// Mitsubishi GX Works2 project: EX2_GROUP21   PLC: FX3G

// global labels: Global1
VAR_GLOBAL
  Emergency AT X005 : BOOL;
  Enough_Materials AT M1 : BOOL;
  Storage_Packs AT D1100 : REAL;
END_VAR
VAR_GLOBAL CONSTANT
  Esroni : REAL := 10.0;
END_VAR
VAR_GLOBAL
  Packs_Display AT D8282 : INT;
  Start_Day AT X007 : BOOL;
  AI_GumType AT D8280 : INT;
  Init_raspberry AT D1150 : REAL;
  Stock_Raspberry AT D2500 : REAL;
  Stock_Lemon AT D2200 : REAL;
  Init_Stabilizer AT D1130 : REAL;
  Stock_Stabilizer AT D2300 : REAL;
  Init_Gummies AT D1140 : REAL;
  Stock_Gummies AT D2400 : REAL;
  Start_Production AT X001 : BOOL;
  Enough_Raspberry AT M9 : BOOL;
  Enough_Lemon AT M10 : BOOL;
  Enough_Stabilizer AT M11 : BOOL;
  Enough_Gummies AT M12 : BOOL;
  Day_Lamp AT Y007 : BOOL;
  GumType_Sempeld AT D3000 : REAL;
  Type_Regular AT M3 : BOOL;
  Type_Premium AT M2 : BOOL;
  Step_Preparation AT M4 : BOOL;
  Prep_Timer AT TC0 : BOOL;
  Stop_Blend AT M14 : BOOL;
  Prep_Counter AT TS0 : BOOL;
  Prep_Lamp AT Y000 : BOOL;
  Start_Cooling AT X002 : BOOL;
  Stop_Prep AT M13 : BOOL;
  Step_Cooling AT M5 : BOOL;
  Stop_Cooling AT TS1 : BOOL;
  Temp_OK AT X003 : BOOL;
  Cooling_Timer AT TC1 : BOOL;
  Cool_Time AT K80 : INT;
  Cooling_Lamp AT Y002 : BOOL;
  Step_Mixing AT M6 : BOOL;
  Blink_Bit AT M8 : BOOL;
  Blink_Time AT K10 : INT;
  Mix_LampA AT Y005 : BOOL;
  Blink_TimerB AT TC3 : BOOL;
  Blink_TimerA AT TC2 : BOOL;
  Stop_BlinkingB AT TS3 : BOOL;
  Stop_BlinkingA AT TS2 : BOOL;
  Mix_LampB AT Y006 : BOOL;
  Mix_Timer_R AT TC4 : BOOL;
  Regular_Mixing_Time AT K30 : INT;
  Mix_Timer_P AT TC5 : BOOL;
  Premium_Mixing_Time AT K50 : INT;
  Mixing_Timer_R AT TS4 : BOOL;
  Mixing_Timer_P AT TS5 : BOOL;
END_VAR
VAR_GLOBAL CONSTANT
  Constant280 : REAL := 280.0;
  Constant400 : REAL := 400.0;
END_VAR
VAR_GLOBAL
  Start_Packing AT M15 : BOOL;
END_VAR
VAR_GLOBAL CONSTANT
  Add_Pack : REAL := 1.0;
  LE_K5 : REAL := 5.0;
  GT_K6 : REAL := 6.0;
  GT_K10 : REAL := 10.0;
  ReqRaspberry : REAL := 385.0;
  ReqLemon : REAL := 665.0;
  ReqStabilizer : REAL := 210.0;
  ReqGummies : REAL := 70.0;
END_VAR
VAR_GLOBAL
  GumType_Final AT D3010 : REAL;
END_VAR
VAR_GLOBAL CONSTANT
  LE_K10 : REAL := 10.0;
END_VAR
VAR_GLOBAL
  Type_R AT M16 : BOOL;
END_VAR
VAR_GLOBAL CONSTANT
  ZeroStartDay : REAL;
END_VAR
VAR_GLOBAL
  Init_Lemon AT D1120 : REAL;
END_VAR
VAR_GLOBAL CONSTANT
  Respberry_280 : REAL := 280.0;
  Gummies_28 : REAL := 28.0;
  Stebilizer_105 : REAL := 105.0;
  Lemon_455 : REAL := 455.0;
END_VAR
VAR_GLOBAL
  Sec_5 AT K50 : INT;
  Not_Active AT M17 : BOOL;
END_VAR

// task Task_01 (event TRUE, interval 0, priority 31): POU_01

PROGRAM POU_01
(* structured ladder/FBD written out as ST: instructions are called as NAME(EN, inputs, outputs); _pN, _eN, _tN stand for wires *)
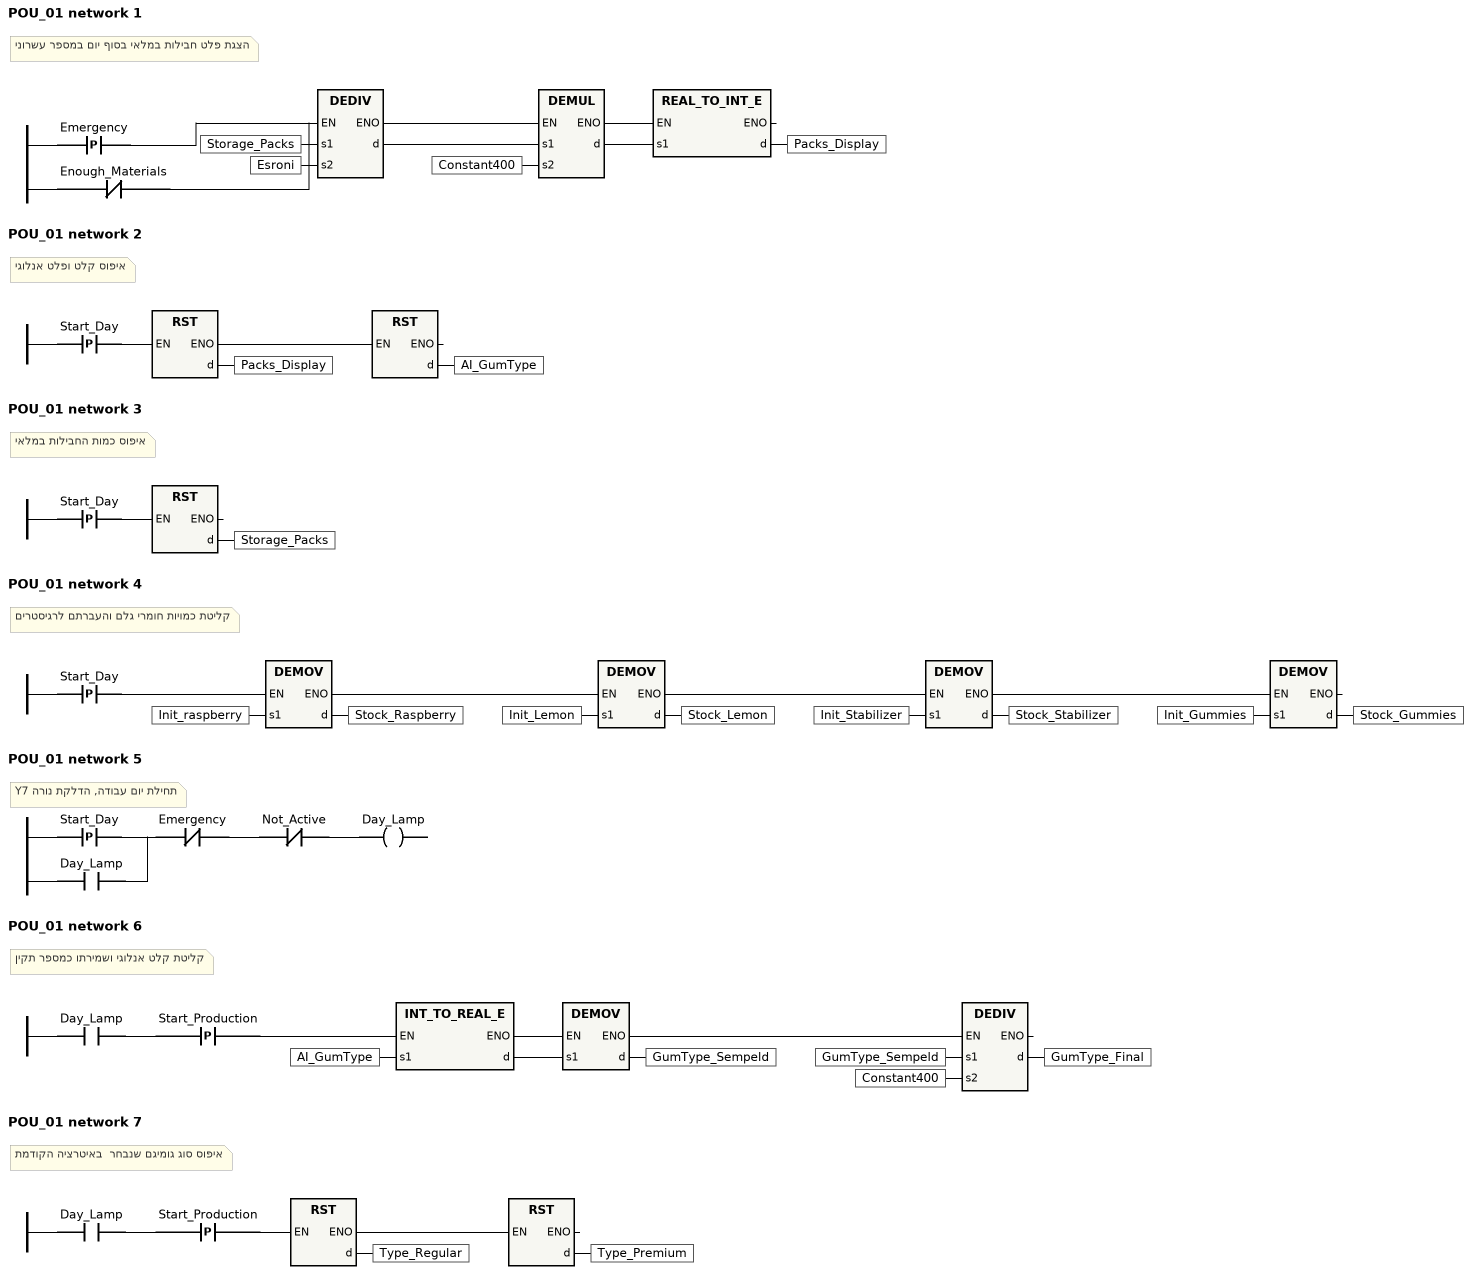
(* network 1 *)
(* הצגת פלט חבילות במלאי בסוף יום במספר עשרוני *)
_e2 := DEDIV(LDP(TRUE, Emergency) OR (NOT Enough_Materials), Storage_Packs, Esroni, _t1);
_e4 := DEMUL(_e2, _t1, Constant400, _t3);
REAL_TO_INT_E(_e4, _t3, Packs_Display);
(* network 2 *)
(* איפוס קלט ופלט אנלוגי *)
_e1 := RST(LDP(TRUE, Start_Day), Packs_Display);
RST(_e1, AI_GumType);
(* network 3 *)
(* איפוס כמות החבילות במלאי *)
RST(LDP(TRUE, Start_Day), Storage_Packs);
(* network 4 *)
(* קליטת כמויות חומרי גלם והעברתם לרגיסטרים *)
_e1 := DEMOV(LDP(TRUE, Start_Day), Init_raspberry, Stock_Raspberry);
_e2 := DEMOV(_e1, Init_Lemon, Stock_Lemon);
_e3 := DEMOV(_e2, Init_Stabilizer, Stock_Stabilizer);
DEMOV(_e3, Init_Gummies, Stock_Gummies);
(* network 5 *)
(* תחילת יום עבודה, הדלקת נורה Y7 *)
Day_Lamp := ((LDP(TRUE, Start_Day) OR Day_Lamp) AND NOT Emergency) AND NOT Not_Active;
(* network 6 *)
(* קליטת קלט אנלוגי ושמירתו כמספר תקין *)
_e2 := INT_TO_REAL_E(Day_Lamp AND LDP(TRUE, Start_Production), AI_GumType, _t1);
_e3 := DEMOV(_e2, _t1, GumType_Sempeld);
DEDIV(_e3, GumType_Sempeld, Constant400, GumType_Final);
(* network 7 *)
(* איפוס סוג גומיגם שנבחר  באיטרציה הקודמת *)
_e1 := RST(Day_Lamp AND LDP(TRUE, Start_Production), Type_Regular);
RST(_e1, Type_Premium);
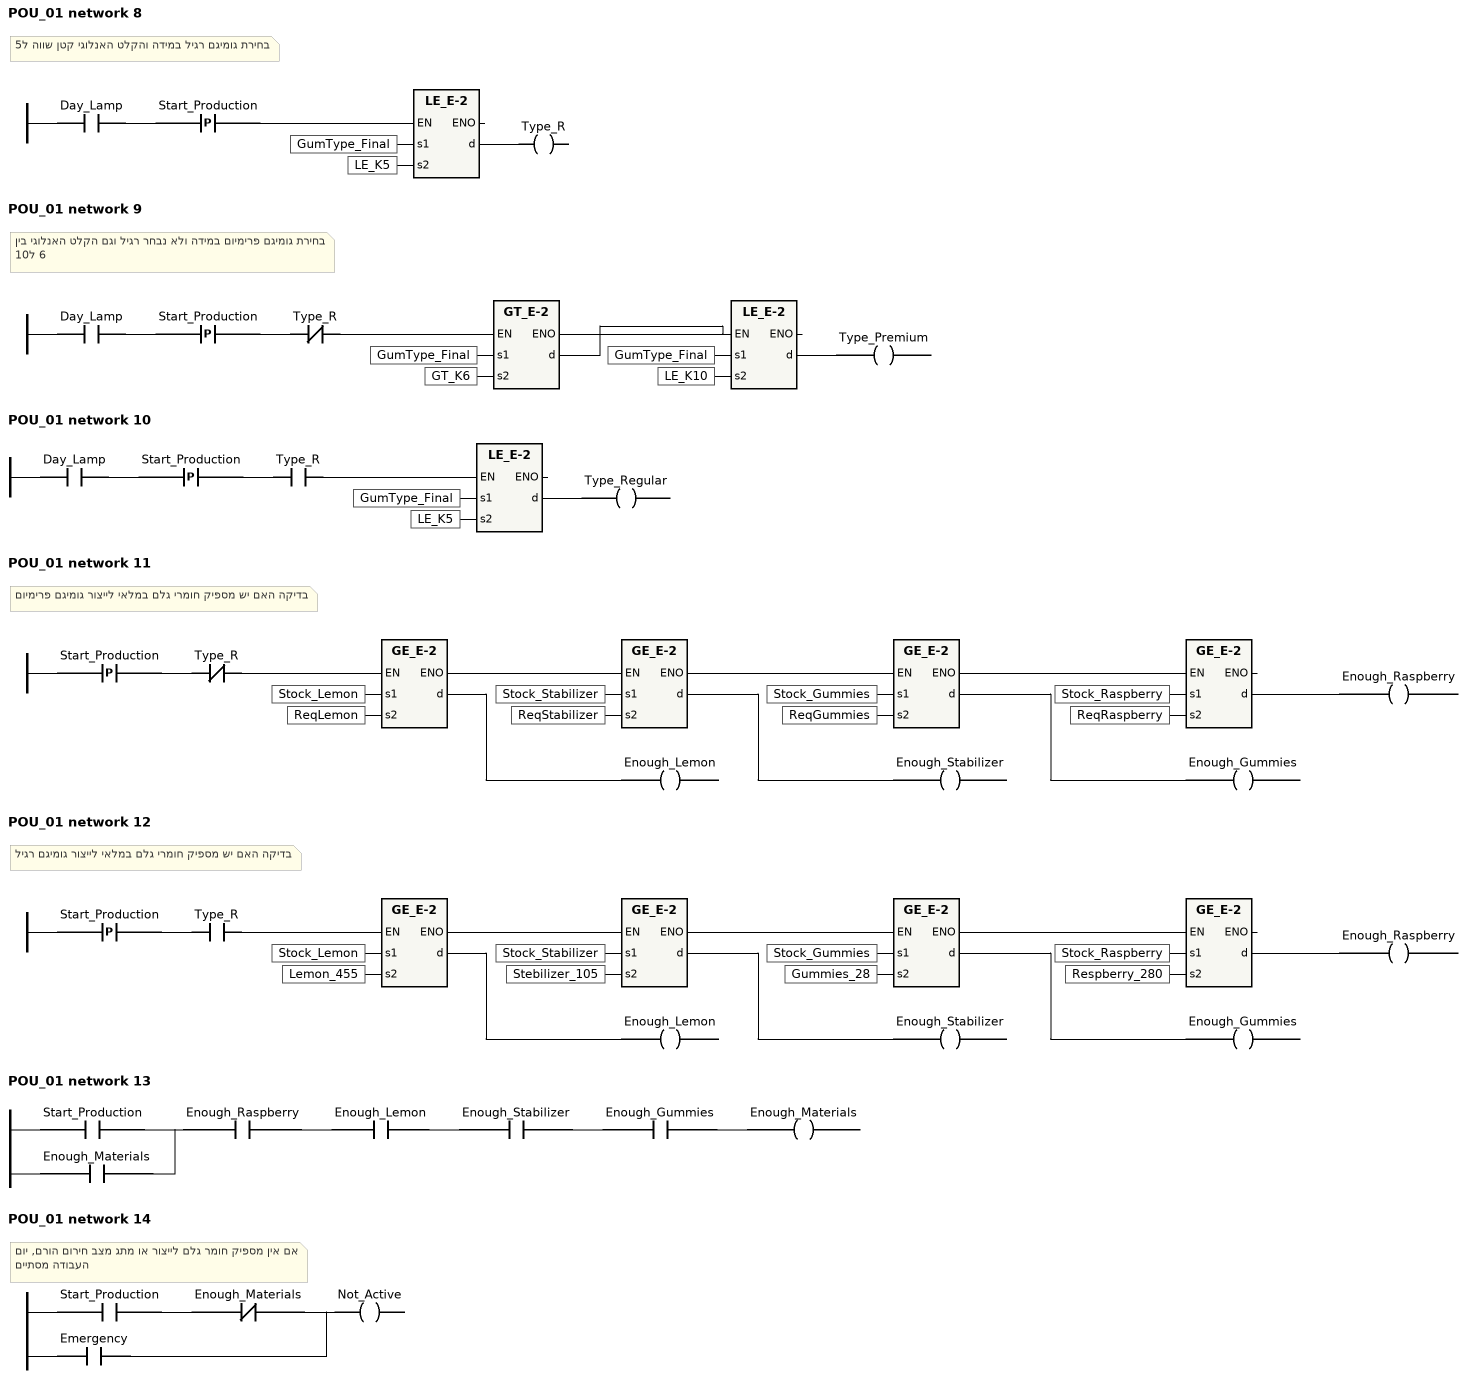
(* network 8 *)
(* בחירת גומיגם רגיל במידה והקלט האנלוגי קטן שווה ל5 *)
LE_E(Day_Lamp AND LDP(TRUE, Start_Production), GumType_Final, LE_K5, _t1);
Type_R := _t1;
(* network 9 *)
(* בחירת גומיגם פרימיום במידה ולא נבחר רגיל וגם הקלט האנלוגי בין 6 ל10 *)
_e2 := GT_E(Day_Lamp AND LDP(TRUE, Start_Production) AND NOT Type_R, GumType_Final, GT_K6, _t1);
LE_E(_e2 OR _t1, GumType_Final, LE_K10, _t3);
Type_Premium := _t3;
(* network 10 *)
LE_E(Day_Lamp AND LDP(TRUE, Start_Production) AND Type_R, GumType_Final, LE_K5, _t1);
Type_Regular := _t1;
(* network 11 *)
(* בדיקה האם יש מספיק חומרי גלם במלאי לייצור גומיגם פרימיום *)
_e2 := GE_E(LDP(TRUE, Start_Production) AND NOT Type_R, Stock_Lemon, ReqLemon, _t1);
_e4 := GE_E(_e2, Stock_Stabilizer, ReqStabilizer, _t3);
_e6 := GE_E(_e4, Stock_Gummies, ReqGummies, _t5);
GE_E(_e6, Stock_Raspberry, ReqRaspberry, _t7);
Enough_Raspberry := _t7;
Enough_Lemon := _t1;
Enough_Stabilizer := _t3;
Enough_Gummies := _t5;
(* network 12 *)
(* בדיקה האם יש מספיק חומרי גלם במלאי לייצור גומיגם רגיל *)
_e2 := GE_E(LDP(TRUE, Start_Production) AND Type_R, Stock_Lemon, Lemon_455, _t1);
_e4 := GE_E(_e2, Stock_Stabilizer, Stebilizer_105, _t3);
_e6 := GE_E(_e4, Stock_Gummies, Gummies_28, _t5);
GE_E(_e6, Stock_Raspberry, Respberry_280, _t7);
Enough_Raspberry := _t7;
Enough_Lemon := _t1;
Enough_Stabilizer := _t3;
Enough_Gummies := _t5;
(* network 13 *)
Enough_Materials := ((((Start_Production OR Enough_Materials) AND Enough_Raspberry) AND Enough_Lemon) AND Enough_Stabilizer) AND Enough_Gummies;
(* network 14 *)
(* אם אין מספיק חומר גלם לייצור או מתג מצב חירום הורם, יום העבודה מסתיים *)
Not_Active := (Start_Production AND NOT Enough_Materials) OR Emergency;
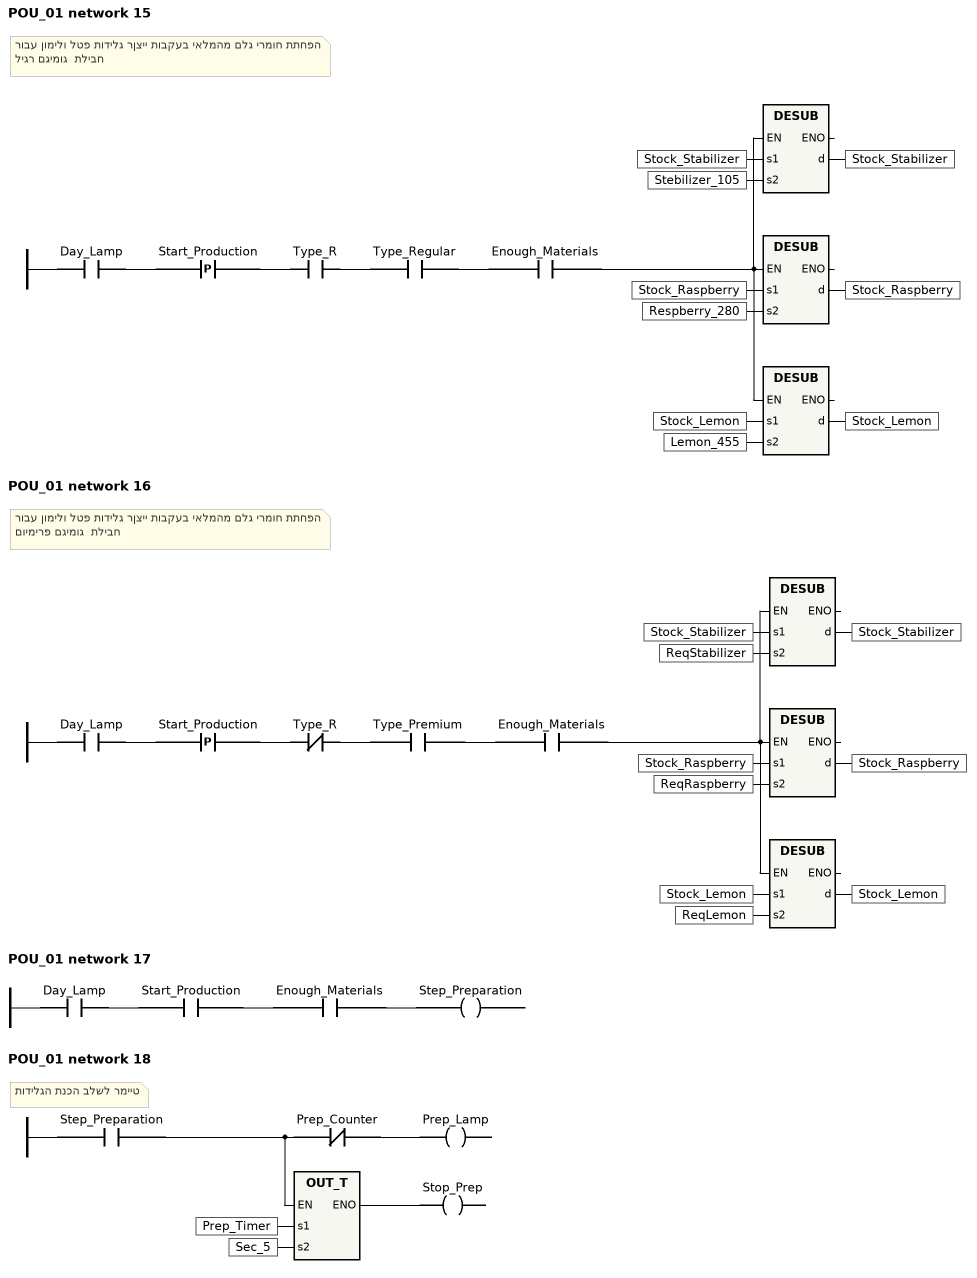
(* network 15 *)
(* הפחתת חומרי גלם מהמלאי בעקבות ייצןר גלידות פטל ולימון עבור חבילת  גומיגם רגיל *)
_p1 := Day_Lamp AND LDP(TRUE, Start_Production) AND Type_R AND Type_Regular AND Enough_Materials;
DESUB(_p1, Stock_Stabilizer, Stebilizer_105, Stock_Stabilizer);
DESUB(_p1, Stock_Raspberry, Respberry_280, Stock_Raspberry);
DESUB(_p1, Stock_Lemon, Lemon_455, Stock_Lemon);
(* network 16 *)
(* הפחתת חומרי גלם מהמלאי בעקבות ייצןר גלידות פטל ולימון עבור חבילת  גומיגם פרימיום *)
_p1 := Day_Lamp AND LDP(TRUE, Start_Production) AND NOT Type_R AND Type_Premium AND Enough_Materials;
DESUB(_p1, Stock_Stabilizer, ReqStabilizer, Stock_Stabilizer);
DESUB(_p1, Stock_Raspberry, ReqRaspberry, Stock_Raspberry);
DESUB(_p1, Stock_Lemon, ReqLemon, Stock_Lemon);
(* network 17 *)
Step_Preparation := Day_Lamp AND Start_Production AND Enough_Materials;
(* network 18 *)
(* טיימר לשלב הכנת הגלידות *)
Prep_Lamp := Step_Preparation AND NOT Prep_Counter;
_e1 := OUT_T(Step_Preparation, Prep_Timer, Sec_5);
Stop_Prep := _e1;
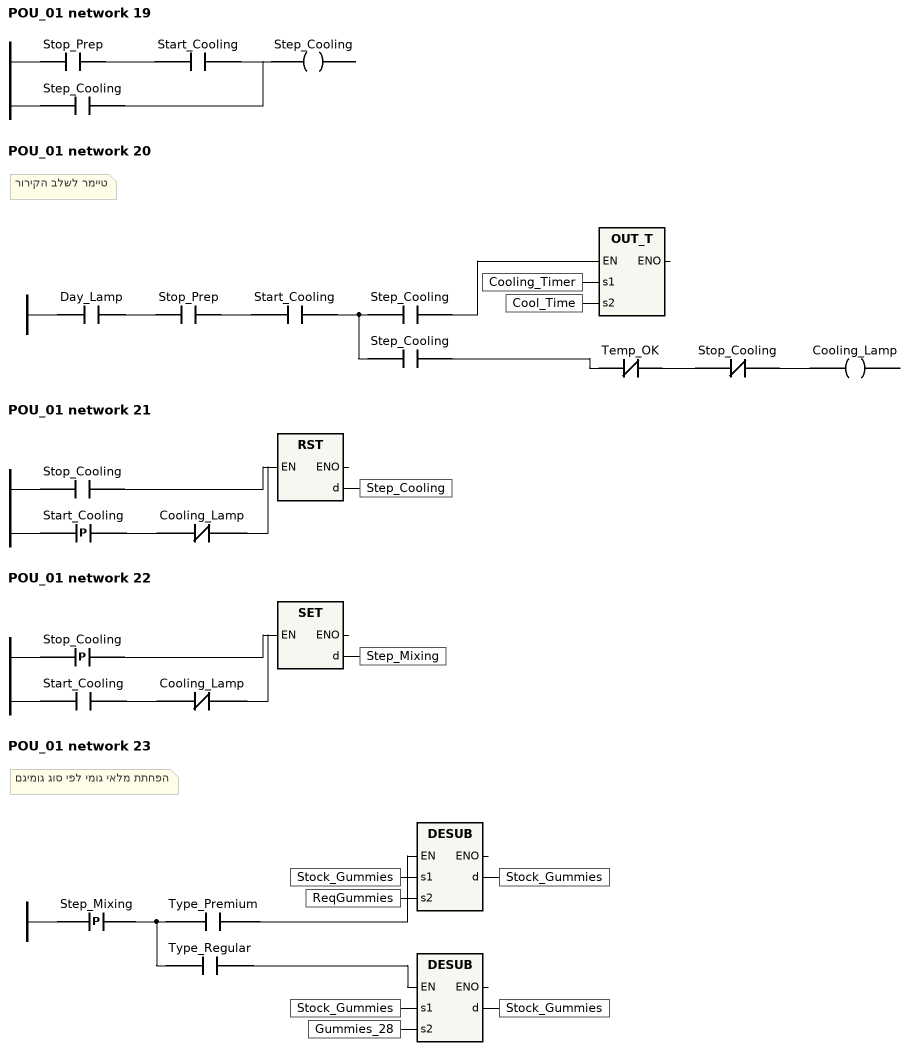
(* network 19 *)
Step_Cooling := (Stop_Prep AND Start_Cooling) OR Step_Cooling;
(* network 20 *)
(* טיימר לשלב הקירור *)
_p1 := Day_Lamp AND Stop_Prep AND Start_Cooling;
OUT_T(_p1 AND Step_Cooling, Cooling_Timer, Cool_Time);
Cooling_Lamp := _p1 AND Step_Cooling AND NOT Temp_OK AND NOT Stop_Cooling;
(* network 21 *)
RST(Stop_Cooling OR (LDP(TRUE, Start_Cooling) AND NOT Cooling_Lamp), Step_Cooling);
(* network 22 *)
SET(LDP(TRUE, Stop_Cooling) OR (Start_Cooling AND NOT Cooling_Lamp), Step_Mixing);
(* network 23 *)
(* הפחתת מלאי גומי לפי סוג גומיגם *)
_p1 := LDP(TRUE, Step_Mixing);
DESUB(_p1 AND Type_Premium, Stock_Gummies, ReqGummies, Stock_Gummies);
DESUB(_p1 AND Type_Regular, Stock_Gummies, Gummies_28, Stock_Gummies);
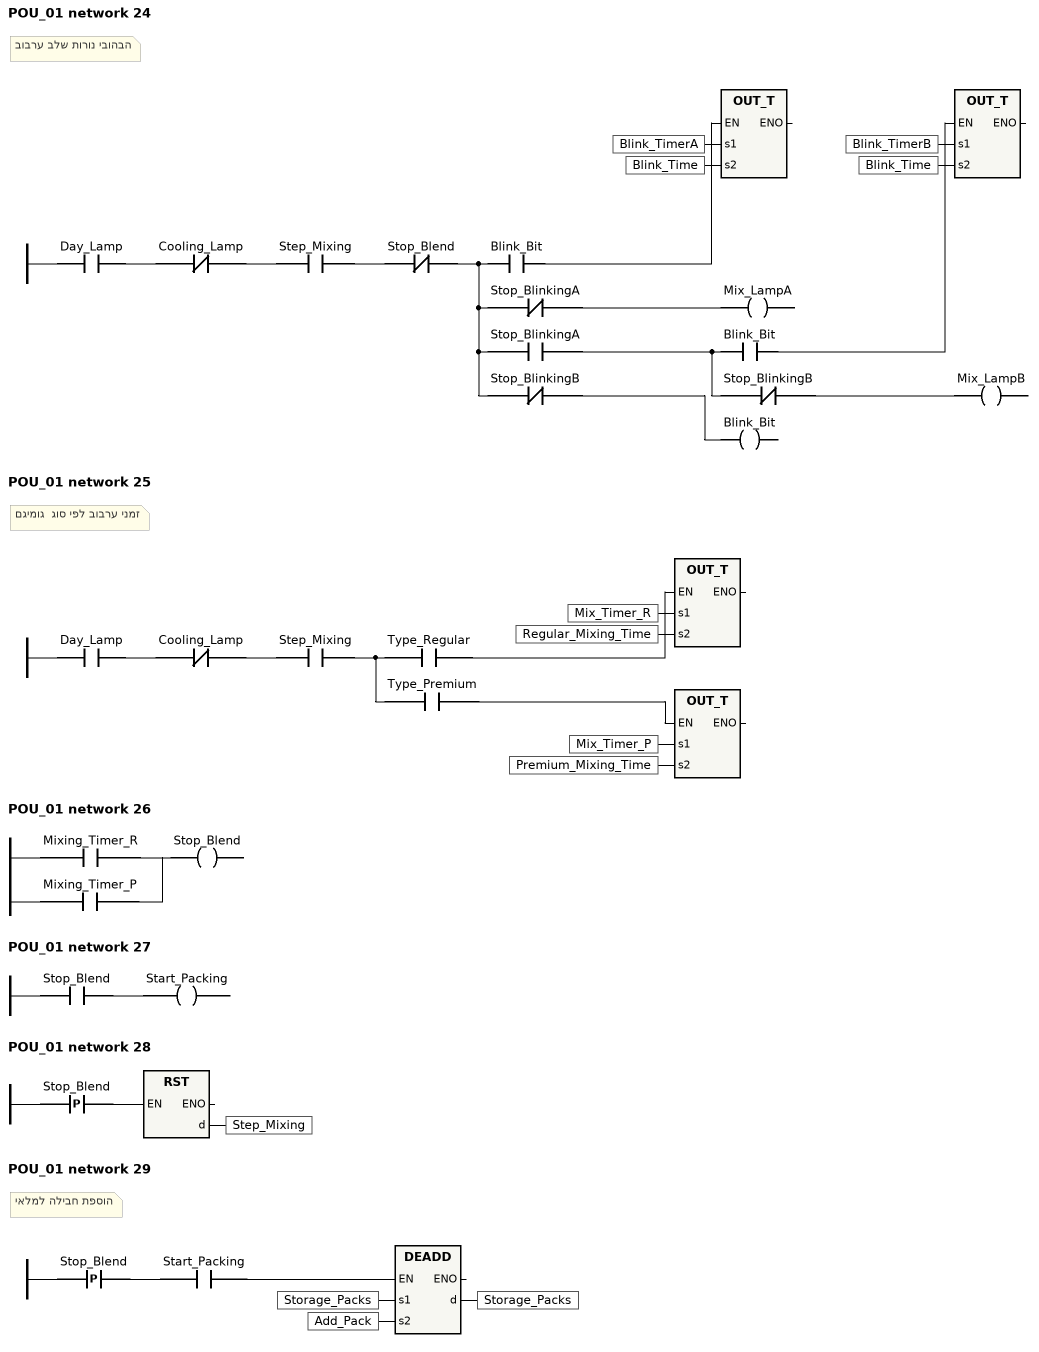
(* network 24 *)
(* הבהובי נורות שלב ערבוב *)
_p1 := Day_Lamp AND NOT Cooling_Lamp AND Step_Mixing AND NOT Stop_Blend;
OUT_T(_p1 AND Blink_Bit, Blink_TimerA, Blink_Time);
Mix_LampA := _p1 AND NOT Stop_BlinkingA;
_p2 := _p1 AND Stop_BlinkingA;
OUT_T(_p2 AND Blink_Bit, Blink_TimerB, Blink_Time);
Mix_LampB := _p2 AND NOT Stop_BlinkingB;
Blink_Bit := _p1 AND NOT Stop_BlinkingB;
(* network 25 *)
(* זמני ערבוב לפי סוג  גומיגם *)
_p1 := Day_Lamp AND NOT Cooling_Lamp AND Step_Mixing;
OUT_T(_p1 AND Type_Regular, Mix_Timer_R, Regular_Mixing_Time);
OUT_T(_p1 AND Type_Premium, Mix_Timer_P, Premium_Mixing_Time);
(* network 26 *)
Stop_Blend := Mixing_Timer_R OR Mixing_Timer_P;
(* network 27 *)
Start_Packing := Stop_Blend;
(* network 28 *)
RST(LDP(TRUE, Stop_Blend), Step_Mixing);
(* network 29 *)
(* הוספת חבילה למלאי *)
DEADD(LDP(TRUE, Stop_Blend) AND Start_Packing, Storage_Packs, Add_Pack, Storage_Packs);
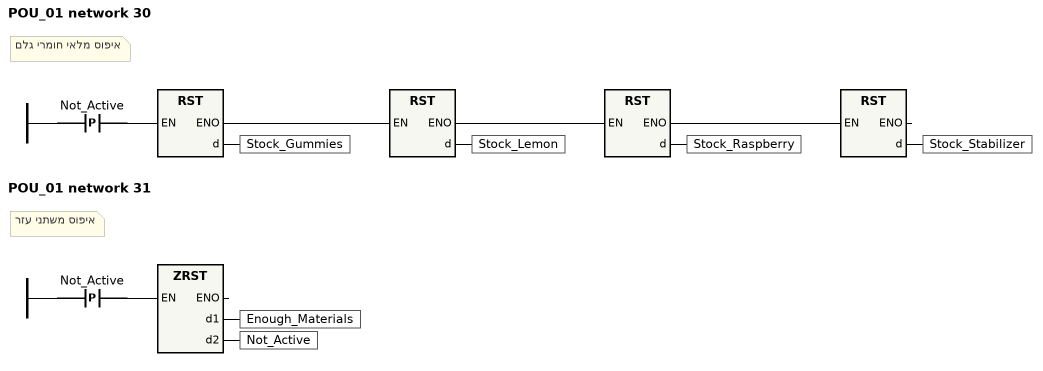
(* network 30 *)
(* איפוס מלאי חומרי גלם *)
_e1 := RST(LDP(TRUE, Not_Active), Stock_Gummies);
_e2 := RST(_e1, Stock_Lemon);
_e3 := RST(_e2, Stock_Raspberry);
RST(_e3, Stock_Stabilizer);
(* network 31 *)
(* איפוס משתני עזר *)
ZRST(LDP(TRUE, Not_Active), Enough_Materials, Not_Active);
END_PROGRAM
